// TIA Portal V16 export
// export: Created 2026-06-22T01:28:19.1477255Z, ExportSetting WithDefaults, DisplayName Totally Integrated Automation Portal, DisplayVersion V16 Update 8, DisplayName TIA Portal Version Control Interface, DisplayVersion V16 Update 8, DisplayName TIA Portal Openness, DisplayVersion V16 Update 8, DisplayName SINAMICS Startdrive Advanced, DisplayVersion V16, DisplayName SINAMICS Startdrive G130, G150, S120, S150, SINAMICS MV, S210, DisplayVersion V16, DisplayName SINAMICS Startdrive G110M, G120, G120C, G120D, G120P, DisplayVersion V16, DisplayName STEP 7 Professional, DisplayVersion V16 Update 8, DisplayName STEP 7 Safety, DisplayVersion V16 Update 7, DisplayName WinCC Advanced, DisplayVersion V16 Update 8
Screen "Motor_Control"  800x480, Number=1
  ScreenLayer 
    Circle "LMP_Run" at 48,176 size 48x48
      RangeAppearanceAnimation "RangeAppearanceAnimation"
        tag STS_Motor_Running
        0..0: back #d9d9d9, fore #181c31
        1..1: back #00ff00, fore #181c31
    Circle "LMP_Fault" at 200,176 size 48x48
      RangeAppearanceAnimation "RangeAppearanceAnimation"
        tag LMP_Motor_Fault
        0..0: back #d9d9d9, fore #181c31
        1..1: back #00ff00, fore #181c31
    Button "BTN_Start" at 24,80 size 110x50  Mode=Text, TextOff="启动", TextOn="启动"
      on Press: SetBit(Tag := BTN_Motor_Start)
      on Release: ResetBit(Tag := BTN_Motor_Start)
    Button "BTN_Reset" at 292,80 size 110x50  Mode=Text, TextOff="复位", TextOn="复位"
      on Press: SetBit(Tag := BTN_Motor_Reset)
      on Release: ResetBit(Tag := BTN_Motor_Reset)
    Button "BTN_Stop" at 158,80 size 110x50  Mode=Text, TextOff="停止", TextOn="停止"
      on Press: SetBit(Tag := BTN_Motor_Stop)
      on Release: ResetBit(Tag := BTN_Motor_Stop)
    IOField "IO_Speed" at 116,268 size 150x40  DataFormat=Decimal, FormatPattern=9999999, Mode=InOutput, ProcessTag=IO_Motor_Speed
    SymbolicIOField "SIO_Mode" at 116,338 size 150x40  CountVisibleItems=3, Mode=InOutput, OnValue=1, ProcessTag=SIO_Motor_Mode, TextOff="0", TextOn="1"
    TextField "TXT_Title" at 200,20 size 400x36  Text="电机控制画面"
    TextField "TXT_ModeLabel" at 24,338 size 80x30  Text="运行模式"
    TextField "TXT_SpeedLabel" at 24,268 size 80x30  Text="转速"
